FUNCTION_BLOCK ContinousSync
VAR_INPUT
	bStart : BOOL; //start the jogging of the master
	bStop : BOOL; //button to stop and reset the movement
END_VAR
VAR_OUTPUT
END_VAR
VAR
	iState : States;	
	
	rSyncPos : LREAL; //position where they sync
	
	fbGetSyncPos : R_TRIG; //we read the sync pos
	fbSyncTimer : TON; //timers that control when the sync and desync start
	fbDesyncTimer : TON;
	
	rActualMasterPos : LREAL; //the actual position of the master axis
	rActualSlavePos : LREAL; //the actual position of the slave axis	
	
	
	MasterAxis : AXIS_REF; //reference to the master and slave axis respectively
	SlaveAxis : AXIS_REF;
	
	PowerMaster : MC_Power; //power function blocks for the master and slave
	PowerSlave : MC_Power; 
	
	ResetMaster : MC_Reset; //reset function blocks for the master and slave
	ResetSlave : MC_Reset; 
	
	StopMaster : MC_Stop; //stop function blocks for the master and slave
	StopSlave : MC_Stop;

	JogMaster : MC_Jog; //function block to move the master
	
	FlyingSaw : MC_GearInPos; //function blocks for gearing in/out
	GearOut : MC_GearOut;
	
	MoveMaster : MC_MoveAbsolute;
	MoveSlave : MC_MoveAbsolute;
		
END_VAR

CASE iState OF
	States.CheckOnline: //check if the axes are turned on
		IF PowerMaster.Enable AND PowerSlave.Enable THEN
			iState := States.StartMaster;
		END_IF
		IF JogMaster.Error THEN
			iState := States.ErrorAndReset; //if an error occurs go to the error handling state
		END_IF
	States.StartMaster: //start the master if the button is pressed
		IF bStart THEN
			JogMaster(Axis := MasterAxis,JogForward := TRUE);
			iState := States.Synchronization;
		END_IF
	States.Synchronization: //start the sync process
		fbGetSyncPos(CLK := FALSE);
		fbSyncTimer.IN := TRUE;
		IF fbSyncTimer.Q THEN
			iState := States.ReadPosition;
		END_IF
		IF JogMaster.Error OR bStop THEN //incase an error or occurs or we stop it manually
			iState := States.ErrorAndReset;			
		END_IF
	States.ReadPosition: //write sync pos
		fbSyncTimer.IN := FALSE;
		fbGetSyncPos(CLK := TRUE); //we read the sync pos
		IF fbGetSyncPos.Q THEN
			rSyncPos := rActualMasterPos + 135.0;
			iState := States.ActivateFlyingSaw; 
		END_IF
		IF JogMaster.Error OR bStop THEN //incase an error or occurs or we stop it manually
			iState := States.ErrorAndReset;			
		END_IF
	States.ActivateFlyingSaw: //flying saw
		fbGetSyncPos(CLK := FALSE);
		FlyingSaw(Master := MasterAxis,Slave := SlaveAxis,MasterSyncPosition := rSyncPos,SlaveSyncPosition := rSyncPos,Execute := TRUE);
		fbDesyncTimer.IN := TRUE; //we start the desync timer
		IF fbDesyncTimer.Q THEN
			iState := States.GearOut;
		END_IF
		IF JogMaster.Error OR bStop THEN //incase an error or occurs or we stop it manually
			iState := States.ErrorAndReset;			
		END_IF
	States.GearOut: //Gear out and stop the slave
		fbDesyncTimer.IN := FALSE;
		StopSlave(Axis := SlaveAxis,Deceleration := 3000,Execute := TRUE);
		GearOut(Slave := SlaveAxis,Execute := TRUE);
		FlyingSaw(Master := MasterAxis,Slave := SlaveAxis,Execute := FALSE);
		IF StopSlave.Done THEN
			iState := States.TempReset; //reset all the blocks
		END_IF
		IF JogMaster.Error OR bStop THEN //incase an error or occurs or we stop it manually
			iState := States.ErrorAndReset;			
		END_IF
	States.TempReset: //reset gear out
		GearOut(Slave := SlaveAxis,Execute := FALSE);
		StopSlave(Axis := SlaveAxis,Execute := FALSE);
		iState := States.Synchronization;
	States.ErrorAndReset: //error and reset state
		GearOut(Slave := SlaveAxis,Execute := TRUE);
		StopSlave(Axis := SlaveAxis,Execute := TRUE);
		StopMaster(Axis := SlaveAxis,Execute := TRUE);
		fbSyncTimer.IN := FALSE;
		fbDesyncTimer.IN := FALSE;
		fbGetSyncPos(CLK := FALSE);
		JogMaster(Axis := MasterAxis,JogForward := FALSE);
		MoveMaster(Axis := MasterAxis,Execute := FALSE);
		MoveSlave(Axis := SlaveAXis,Execute := FALSE);
		IF JogMaster.Error OR MoveMaster.Error OR MoveSlave.Error THEN
			ResetMaster(Axis := MasterAxis,Execute := TRUE);
			ResetSlave(Axis := SlaveAxis,Execute := TRUE);
		ELSE
			iState := States.ReturnToPosition0; //return to the starting point
		END_IF

	States.ReturnToPosition0: //return to position 0
		GearOut(Slave := SlaveAxis,Execute := FALSE);
		StopSlave(Axis := SlaveAxis,Execute := FALSE);
		StopMaster(Axis := SlaveAxis,Execute := FALSE);
		ResetMaster(Axis := MasterAxis,Execute := FALSE);
		ResetSlave(Axis := SlaveAxis,Execute := FALSE);
		MoveMaster(Axis := MasterAxis,Position := 0,Velocity := 800,Execute := TRUE);
		MoveSlave(Axis := SlaveAxis,Position := 0,Velocity := 800,Execute := TRUE);
		IF MoveMaster.Done AND MoveSlave.Done THEN
			MoveMaster(Axis := MasterAxis,Execute := FALSE);
			MoveSlave(Axis := SlaveAxis,Execute := FALSE);
			iState := 10; //return to the start
		ELSIF MoveMaster.Error OR MoveSlave.Error THEN
			iState := States.ErrorAndReset;
		END_IF
						
END_CASE


PowerMaster(Axis := MasterAxis,Enable := TRUE,Enable_Positive := TRUE,Enable_Negative := TRUE);
PowerSlave(Axis := SlaveAxis,Enable := TRUE,Enable_Positive := TRUE,Enable_Negative := TRUE);

ResetMaster(Axis := MasterAxis);
ResetSlave(Axis := SlaveAxis);

StopMaster(Axis := MasterAxis);
StopSlave(Axis := SlaveAxis);

JogMaster(Axis := MasterAxis);

MoveMaster(Axis := MasterAxis);
MoveSlave(Axis := SlaveAXis);

fbSyncTimer(PT := T#4000MS);
fbDesyncTimer(PT := T#4000MS);

rActualMasterPos := MasterAxis.NcToPlc.ActPos;
rActualSlavePos := SlaveAxis.NcToPlc.ActPos;

END_FUNCTION_BLOCK

(* stored: Version 1.1.0.1, ProductVersion 3.1.4024.12
   POU ContinousSync: Id {d492fa16-1da2-4236-b22a-fe2d8c7710c5}, SpecialFunc None *)
